// TIA Portal V21 export
TYPE "Std_Utente"
   STRUCT
      User : String[10];
      Psw : String[10];
      Livello : Int;
      TimeOut : Real;
   END_STRUCT;
END_TYPE
